FUNCTION_BLOCK FB_TransmitStatesToHMI
VAR_INPUT
END_VAR
VAR_OUTPUT
END_VAR
VAR
	fSetAlarm : FB_SetAlarm;
END_VAR

// safeties
GVL_HMI.i_b24VDC_CB_OK := GVL_IO.DI_24VDC_CB_OK;
IF NOT GVL_HMI.i_b24VDC_CB_OK THEN
	fSetAlarm( sMsg := GVL_AlarmMessage.DC_FAIL );
END_IF
GVL_HMI.i_bESR1 := GVL_IO.DI_ESR1;
IF NOT GVL_HMI.i_bESR1 THEN
	fSetAlarm( sMsg := GVL_AlarmMessage.ESR1_FAIL );
END_IF
GVL_HMI.i_bLS1 := GVL_IO.DI_LS1;
GVL_HMI.i_bTS1 := GVL_IO.DI_TS1;
GVL_HMI.i_bPS1 := GVL_IO.DI_PS1;

// Output
GVL_HMI.i_bVB1 := GVL_IO.DO_VB1;
GVL_HMI.i_bVB2 := GVL_IO.DO_VB2;
GVL_HMI.i_bCyl1E := GVL_IO.DO_CYL1_E;
GVL_HMI.i_bCyl1R := GVL_IO.DO_CYL1_R;
GVL_HMI.i_bCyl2E := GVL_IO.DO_CYL2_E;
GVL_HMI.i_bCyl2R := GVL_IO.DO_CYL2_R;
GVL_HMI.i_bCyl3E := GVL_IO.DO_CYL3_E;
GVL_HMI.i_bCyl3R := GVL_IO.DO_CYL3_R;
GVL_HMI.i_bCyl4E := GVL_IO.DO_CYL4_E;
GVL_HMI.i_bCyl4R := GVL_IO.DO_CYL4_R;
GVL_HMI.i_bCyl5E := GVL_IO.DO_CYL5_E;
GVL_HMI.i_bCyl5R := GVL_IO.DO_CYL5_R;
GVL_HMI.i_bCyl6E := GVL_IO.DO_CYL6_E;
GVL_HMI.i_bCyl6R := GVL_IO.DO_CYL6_R;
GVL_HMI.i_bCyl7E := GVL_IO.DO_CYL7_E;
GVL_HMI.i_bCyl7R := GVL_IO.DO_CYL7_R;
GVL_HMI.i_bCyl8E := GVL_IO.DO_CYL8_E;
GVL_HMI.i_bCyl8R := GVL_IO.DO_CYL8_R;

// Vibratory
GVL_HMI.i_bPE1 := GVL_IO.DI_PE1;
IF NOT GVL_HMI.i_bPE1 THEN
	fSetAlarm( sMsg := GVL_AlarmMessage.PE1_FAIL );
END_IF
GVL_HMI.i_bPE2 := GVL_IO.DI_PE2;
IF NOT GVL_HMI.i_bPE2 THEN
	fSetAlarm( sMsg := GVL_AlarmMessage.PE2_FAIL );
END_IF
GVL_HMI.i_bPE3 := GVL_IO.DI_PE3;
IF NOT GVL_HMI.i_bPE3 THEN
	fSetAlarm( sMsg := GVL_AlarmMessage.PE3_FAIL );
END_IF
GVL_HMI.i_bPE4 := GVL_IO.DI_PE4;
IF NOT GVL_HMI.i_bPE4 THEN
	fSetAlarm( sMsg := GVL_AlarmMessage.PE4_FAIL );
END_IF
GVL_HMI.i_bPE5 := GVL_IO.DI_PE5;
IF NOT GVL_HMI.i_bPE5 THEN
	fSetAlarm( sMsg := GVL_AlarmMessage.PE5_FAIL );
END_IF

// analog value
GVL_HMI.i_rPT1 := GVL_IO.AI_PT1;
GVL_HMI.i_rPT2 := GVL_IO.AI_PT2;

// enabling flag
GVL_HMI.i_bECS := GVL_IO.DI_ECS;

// led
IF NOT GVL_HMI.o_bAlarmActive THEN
	GVL_IO.DO_LGreen := FALSE;
	GVL_IO.DO_LRed := TRUE;
ELSE
	GVL_IO.DO_LGreen := TRUE;
	GVL_IO.DO_LRed := FALSE;
END_IF

IF (GVL_HMI.i_nCylinder1State>=0) OR (GVL_HMI.i_nCylinder1State MOD 2 = 0) THEN
	IF GVL_IO.DI_CYL1_E THEN GVL_HMI.i_nCylinder1State := 0; ELSIF GVL_IO.DI_CYL1_R THEN GVL_HMI.i_nCylinder1State := 2; END_IF
END_IF
IF (GVL_HMI.i_nCylinder2State>=0) OR (GVL_HMI.i_nCylinder2State MOD 2 = 0) THEN
	IF GVL_IO.DI_CYL2_E THEN GVL_HMI.i_nCylinder2State := 0; ELSIF GVL_IO.DI_CYL2_R THEN GVL_HMI.i_nCylinder2State := 2; END_IF
END_IF
IF (GVL_HMI.i_nCylinder3State>=0) OR (GVL_HMI.i_nCylinder3State MOD 2 = 0) THEN
	IF GVL_IO.DI_CYL3_E THEN GVL_HMI.i_nCylinder3State := 0; ELSIF GVL_IO.DI_CYL3_R THEN GVL_HMI.i_nCylinder3State := 2; END_IF
END_IF
IF (GVL_HMI.i_nCylinder4State>=0) OR (GVL_HMI.i_nCylinder4State MOD 2 = 0) THEN
	IF GVL_IO.DI_CYL4_E THEN GVL_HMI.i_nCylinder4State := 0; ELSIF GVL_IO.DI_CYL4_R THEN GVL_HMI.i_nCylinder4State := 2; END_IF
END_IF
IF (GVL_HMI.i_nCylinder5State>=0) OR (GVL_HMI.i_nCylinder5State MOD 2 = 0) THEN
	IF GVL_IO.DI_CYL5_E THEN GVL_HMI.i_nCylinder5State := 0; ELSIF GVL_IO.DI_CYL5_R THEN GVL_HMI.i_nCylinder5State := 2; END_IF
END_IF
IF (GVL_HMI.i_nCylinder6State>=0) OR (GVL_HMI.i_nCylinder6State MOD 2 = 0) THEN
	IF GVL_IO.DI_CYL6_E THEN GVL_HMI.i_nCylinder6State := 0; ELSIF GVL_IO.DI_CYL6_R THEN GVL_HMI.i_nCylinder6State := 2; END_IF
END_IF
IF (GVL_HMI.i_nCylinder7State>=0) OR (GVL_HMI.i_nCylinder7State MOD 2 = 0) THEN
	IF GVL_IO.DI_CYL7_E THEN GVL_HMI.i_nCylinder7State := 0; ELSIF GVL_IO.DI_CYL7_R THEN GVL_HMI.i_nCylinder7State := 2; END_IF
END_IF

END_FUNCTION_BLOCK

(* stored: Version 1.1.0.1, ProductVersion 3.1.4024.6
   POU FB_TransmitStatesToHMI: Id {bd67aa5a-e740-41f9-a2ca-e2a51652f913}, SpecialFunc None *)
